PROGRAM MAIN
VAR
	ccs_sim:	FB_CCS_SIM;
	fbTimer: FB_TIME;
END_VAR

fbTimer();
ccs_sim();

END_PROGRAM

(* stored: Version 1.1.0.1, ProductVersion 3.1.4024.9
   POU MAIN: Id {9341b6a9-ab47-4021-8934-6cc66bcac750}, SpecialFunc None *)
